	RoomTemp_204: FB_BACnetRM_AI := (Client:=Client,nObjectInstance:=52233);
	TempAdjust_204: FB_BACnetRM_AV := (Client:=Client,nObjectInstance:=52234);
	FilterSign_204: FB_BACnetRM_BI := (Client:=Client,nObjectInstance:=52235);
	FilterSignReset_204: FB_BACnetRM_BV := (Client:=Client,nObjectInstance:=52236);
	RemoteControlStart_204: FB_BACnetRM_BV := (Client:=Client,nObjectInstance:=52237);
	
	RemoteControlTempAdjust_204: FB_BACnetRM_BV := (Client:=Client,nObjectInstance:=52240);
	
	
	
	
	
	
	
	
	
	
	
	
	StartStopCommand_205: FB_BACnetRM_BO := (Client:=Client,nObjectInstance:=52481);
	StartStopStatus_205: FB_BACnetRM_BI := (Client:=Client,nObjectInstance:=52482);
	Alarm_205: FB_BACnetRM_BI := (Client:=Client,nObjectInstance:=52483);
	MalfunctionCode_205: FB_BACnetRM_MI := (Client:=Client,nObjectInstance:=52484);
	
	
	
	
	RoomTemp_205: FB_BACnetRM_AI := (Client:=Client,nObjectInstance:=52489);
	TempAdjust_205: FB_BACnetRM_AV := (Client:=Client,nObjectInstance:=52490);
	FilterSign_205: FB_BACnetRM_BI := (Client:=Client,nObjectInstance:=52491);
	FilterSignReset_205: FB_BACnetRM_BV := (Client:=Client,nObjectInstance:=52492);
	RemoteControlStart_205: FB_BACnetRM_BV := (Client:=Client,nObjectInstance:=52493);
	
	RemoteControlTempAdjust_205: FB_BACnetRM_BV := (Client:=Client,nObjectInstance:=52496);
	
	
	
	
	
	
	
	
	
	
	
	
	StartStopCommand_206: FB_BACnetRM_BO := (Client:=Client,nObjectInstance:=52737);
	StartStopStatus_206: FB_BACnetRM_BI := (Client:=Client,nObjectInstance:=52738);
	Alarm_206: FB_BACnetRM_BI := (Client:=Client,nObjectInstance:=52739);
	MalfunctionCode_206: FB_BACnetRM_MI := (Client:=Client,nObjectInstance:=52740);
	
	
	
	
	RoomTemp_206: FB_BACnetRM_AI := (Client:=Client,nObjectInstance:=52745);
	TempAdjust_206: FB_BACnetRM_AV := (Client:=Client,nObjectInstance:=52746);
	FilterSign_206: FB_BACnetRM_BI := (Client:=Client,nObjectInstance:=52747);
	FilterSignReset_206: FB_BACnetRM_BV := (Client:=Client,nObjectInstance:=52748);
	RemoteControlStart_206: FB_BACnetRM_BV := (Client:=Client,nObjectInstance:=52749);
	
	RemoteControlTempAdjust_206: FB_BACnetRM_BV := (Client:=Client,nObjectInstance:=52752);
	
	
	
	
	
	
	
	
	
	
	
	
	StartStopCommand_207: FB_BACnetRM_BO := (Client:=Client,nObjectInstance:=52993);
	StartStopStatus_207: FB_BACnetRM_BI := (Client:=Client,nObjectInstance:=52994);
	Alarm_207: FB_BACnetRM_BI := (Client:=Client,nObjectInstance:=52995);
	MalfunctionCode_207: FB_BACnetRM_MI := (Client:=Client,nObjectInstance:=52996);
	
	
	
	
	RoomTemp_207: FB_BACnetRM_AI := (Client:=Client,nObjectInstance:=53001);
	TempAdjust_207: FB_BACnetRM_AV := (Client:=Client,nObjectInstance:=53002);
	FilterSign_207: FB_BACnetRM_BI := (Client:=Client,nObjectInstance:=53003);
	FilterSignReset_207: FB_BACnetRM_BV := (Client:=Client,nObjectInstance:=53004);
	RemoteControlStart_207: FB_BACnetRM_BV := (Client:=Client,nObjectInstance:=53005);
	
	RemoteControlTempAdjust_207: FB_BACnetRM_BV := (Client:=Client,nObjectInstance:=53008);
	
	
	
	
	
	
	
	
	
	
	
	
	StartStopCommand_208: FB_BACnetRM_BO := (Client:=Client,nObjectInstance:=53249);
	StartStopStatus_208: FB_BACnetRM_BI := (Client:=Client,nObjectInstance:=53250);
	Alarm_208: FB_BACnetRM_BI := (Client:=Client,nObjectInstance:=53251);
	MalfunctionCode_208: FB_BACnetRM_MI := (Client:=Client,nObjectInstance:=53252);
	
	
	
	
	RoomTemp_208: FB_BACnetRM_AI := (Client:=Client,nObjectInstance:=53257);
	TempAdjust_208: FB_BACnetRM_AV := (Client:=Client,nObjectInstance:=53258);
	FilterSign_208: FB_BACnetRM_BI := (Client:=Client,nObjectInstance:=53259);
	FilterSignReset_208: FB_BACnetRM_BV := (Client:=Client,nObjectInstance:=53260);
	RemoteControlStart_208: FB_BACnetRM_BV := (Client:=Client,nObjectInstance:=53261);
	
	RemoteControlTempAdjust_208: FB_BACnetRM_BV := (Client:=Client,nObjectInstance:=53264);
	
	
	
	
	
	
	
	
	
	
	
	
	StartStopCommand_209: FB_BACnetRM_BO := (Client:=Client,nObjectInstance:=53505);
	StartStopStatus_209: FB_BACnetRM_BI := (Client:=Client,nObjectInstance:=53506);
	Alarm_209: FB_BACnetRM_BI := (Client:=Client,nObjectInstance:=53507);
	MalfunctionCode_209: FB_BACnetRM_MI := (Client:=Client,nObjectInstance:=53508);
	
	
	
	
	RoomTemp_209: FB_BACnetRM_AI := (Client:=Client,nObjectInstance:=53513);
	TempAdjust_209: FB_BACnetRM_AV := (Client:=Client,nObjectInstance:=53514);
	FilterSign_209: FB_BACnetRM_BI := (Client:=Client,nObjectInstance:=53515);
	FilterSignReset_209: FB_BACnetRM_BV := (Client:=Client,nObjectInstance:=53516);
	RemoteControlStart_209: FB_BACnetRM_BV := (Client:=Client,nObjectInstance:=53517);
	
	RemoteControlTempAdjust_209: FB_BACnetRM_BV := (Client:=Client,nObjectInstance:=53520);
	
	
	
	
	
	
	
	
	
	
	
	
	StartStopCommand_210: FB_BACnetRM_BO := (Client:=Client,nObjectInstance:=53761);
	StartStopStatus_210: FB_BACnetRM_BI := (Client:=Client,nObjectInstance:=53762);
	Alarm_210: FB_BACnetRM_BI := (Client:=Client,nObjectInstance:=53763);
	MalfunctionCode_210: FB_BACnetRM_MI := (Client:=Client,nObjectInstance:=53764);
	
	
	
	
	RoomTemp_210: FB_BACnetRM_AI := (Client:=Client,nObjectInstance:=53769);
	TempAdjust_210: FB_BACnetRM_AV := (Client:=Client,nObjectInstance:=53770);
	FilterSign_210: FB_BACnetRM_BI := (Client:=Client,nObjectInstance:=53771);
	FilterSignReset_210: FB_BACnetRM_BV := (Client:=Client,nObjectInstance:=53772);
	RemoteControlStart_210: FB_BACnetRM_BV := (Client:=Client,nObjectInstance:=53773);
	
	RemoteControlTempAdjust_210: FB_BACnetRM_BV := (Client:=Client,nObjectInstance:=53776);
	
	
	
	
	
	
	
	
	
	
	
	
	StartStopCommand_211: FB_BACnetRM_BO := (Client:=Client,nObjectInstance:=54017);
	StartStopStatus_211: FB_BACnetRM_BI := (Client:=Client,nObjectInstance:=54018);
	Alarm_211: FB_BACnetRM_BI := (Client:=Client,nObjectInstance:=54019);
	MalfunctionCode_211: FB_BACnetRM_MI := (Client:=Client,nObjectInstance:=54020);
	
	
	
	
	RoomTemp_211: FB_BACnetRM_AI := (Client:=Client,nObjectInstance:=54025);
	TempAdjust_211: FB_BACnetRM_AV := (Client:=Client,nObjectInstance:=54026);
	FilterSign_211: FB_BACnetRM_BI := (Client:=Client,nObjectInstance:=54027);
	FilterSignReset_211: FB_BACnetRM_BV := (Client:=Client,nObjectInstance:=54028);
	RemoteControlStart_211: FB_BACnetRM_BV := (Client:=Client,nObjectInstance:=54029);
	
	RemoteControlTempAdjust_211: FB_BACnetRM_BV := (Client:=Client,nObjectInstance:=54032);
	
	
	
	
	
	
	
	
	
	
	
	
	StartStopCommand_212: FB_BACnetRM_BO := (Client:=Client,nObjectInstance:=54273);
	StartStopStatus_212: FB_BACnetRM_BI := (Client:=Client,nObjectInstance:=54274);
	Alarm_212: FB_BACnetRM_BI := (Client:=Client,nObjectInstance:=54275);
	MalfunctionCode_212: FB_BACnetRM_MI := (Client:=Client,nObjectInstance:=54276);
	
	
	
	
	RoomTemp_212: FB_BACnetRM_AI := (Client:=Client,nObjectInstance:=54281);
	TempAdjust_212: FB_BACnetRM_AV := (Client:=Client,nObjectInstance:=54282);
	FilterSign_212: FB_BACnetRM_BI := (Client:=Client,nObjectInstance:=54283);
	FilterSignReset_212: FB_BACnetRM_BV := (Client:=Client,nObjectInstance:=54284);
	RemoteControlStart_212: FB_BACnetRM_BV := (Client:=Client,nObjectInstance:=54285);
	
	RemoteControlTempAdjust_212: FB_BACnetRM_BV := (Client:=Client,nObjectInstance:=54288);
	
	
	
	
	
	
	
	
	
	
	
	
	StartStopCommand_213: FB_BACnetRM_BO := (Client:=Client,nObjectInstance:=54529);
	StartStopStatus_213: FB_BACnetRM_BI := (Client:=Client,nObjectInstance:=54530);
	Alarm_213: FB_BACnetRM_BI := (Client:=Client,nObjectInstance:=54531);
	MalfunctionCode_213: FB_BACnetRM_MI := (Client:=Client,nObjectInstance:=54532);
	
	
	
	
	RoomTemp_213: FB_BACnetRM_AI := (Client:=Client,nObjectInstance:=54537);
	TempAdjust_213: FB_BACnetRM_AV := (Client:=Client,nObjectInstance:=54538);
	FilterSign_213: FB_BACnetRM_BI := (Client:=Client,nObjectInstance:=54539);
	FilterSignReset_213: FB_BACnetRM_BV := (Client:=Client,nObjectInstance:=54540);
	RemoteControlStart_213: FB_BACnetRM_BV := (Client:=Client,nObjectInstance:=54541);
	
	RemoteControlTempAdjust_213: FB_BACnetRM_BV := (Client:=Client,nObjectInstance:=54544);
	
	
	
	
	
	
	
	
	
	
	
	
	StartStopCommand_214: FB_BACnetRM_BO := (Client:=Client,nObjectInstance:=54785);
	StartStopStatus_214: FB_BACnetRM_BI := (Client:=Client,nObjectInstance:=54786);
	Alarm_214: FB_BACnetRM_BI := (Client:=Client,nObjectInstance:=54787);
	MalfunctionCode_214: FB_BACnetRM_MI := (Client:=Client,nObjectInstance:=54788);
	
	
	
	
	RoomTemp_214: FB_BACnetRM_AI := (Client:=Client,nObjectInstance:=54793);
	TempAdjust_214: FB_BACnetRM_AV := (Client:=Client,nObjectInstance:=54794);
	FilterSign_214: FB_BACnetRM_BI := (Client:=Client,nObjectInstance:=54795);
	FilterSignReset_214: FB_BACnetRM_BV := (Client:=Client,nObjectInstance:=54796);
	RemoteControlStart_214: FB_BACnetRM_BV := (Client:=Client,nObjectInstance:=54797);
	
	RemoteControlTempAdjust_214: FB_BACnetRM_BV := (Client:=Client,nObjectInstance:=54800);
	
	
	
	
	
	
	
	
	
	
	
	
	StartStopCommand_215: FB_BACnetRM_BO := (Client:=Client,nObjectInstance:=55041);
	StartStopStatus_215: FB_BACnetRM_BI := (Client:=Client,nObjectInstance:=55042);
	Alarm_215: FB_BACnetRM_BI := (Client:=Client,nObjectInstance:=55043);
	MalfunctionCode_215: FB_BACnetRM_MI := (Client:=Client,nObjectInstance:=55044);
	
	
	
	
	RoomTemp_215: FB_BACnetRM_AI := (Client:=Client,nObjectInstance:=55049);
	TempAdjust_215: FB_BACnetRM_AV := (Client:=Client,nObjectInstance:=55050);
	FilterSign_215: FB_BACnetRM_BI := (Client:=Client,nObjectInstance:=55051);
	FilterSignReset_215: FB_BACnetRM_BV := (Client:=Client,nObjectInstance:=55052);
	RemoteControlStart_215: FB_BACnetRM_BV := (Client:=Client,nObjectInstance:=55053);
	
	RemoteControlTempAdjust_215: FB_BACnetRM_BV := (Client:=Client,nObjectInstance:=55056);
	
	
	
	
	
	
	
	
	
	
	
	
	StartStopCommand_216: FB_BACnetRM_BO := (Client:=Client,nObjectInstance:=55297);
	StartStopStatus_216: FB_BACnetRM_BI := (Client:=Client,nObjectInstance:=55298);
	Alarm_216: FB_BACnetRM_BI := (Client:=Client,nObjectInstance:=55299);
	MalfunctionCode_216: FB_BACnetRM_MI := (Client:=Client,nObjectInstance:=55300);
	
	
	
	
	RoomTemp_216: FB_BACnetRM_AI := (Client:=Client,nObjectInstance:=55305);
	TempAdjust_216: FB_BACnetRM_AV := (Client:=Client,nObjectInstance:=55306);
	FilterSign_216: FB_BACnetRM_BI := (Client:=Client,nObjectInstance:=55307);
	FilterSignReset_216: FB_BACnetRM_BV := (Client:=Client,nObjectInstance:=55308);
	RemoteControlStart_216: FB_BACnetRM_BV := (Client:=Client,nObjectInstance:=55309);
	
	RemoteControlTempAdjust_216: FB_BACnetRM_BV := (Client:=Client,nObjectInstance:=55312);
	
	
	
	
	
	
	
	
	
	
	
	
	StartStopCommand_217: FB_BACnetRM_BO := (Client:=Client,nObjectInstance:=55553);
	StartStopStatus_217: FB_BACnetRM_BI := (Client:=Client,nObjectInstance:=55554);
	Alarm_217: FB_BACnetRM_BI := (Client:=Client,nObjectInstance:=55555);
	MalfunctionCode_217: FB_BACnetRM_MI := (Client:=Client,nObjectInstance:=55556);
	
	
	
	
	RoomTemp_217: FB_BACnetRM_AI := (Client:=Client,nObjectInstance:=55561);
	TempAdjust_217: FB_BACnetRM_AV := (Client:=Client,nObjectInstance:=55562);
	FilterSign_217: FB_BACnetRM_BI := (Client:=Client,nObjectInstance:=55563);
	FilterSignReset_217: FB_BACnetRM_BV := (Client:=Client,nObjectInstance:=55564);
	RemoteControlStart_217: FB_BACnetRM_BV := (Client:=Client,nObjectInstance:=55565);
	
	RemoteControlTempAdjust_217: FB_BACnetRM_BV := (Client:=Client,nObjectInstance:=55568);
	
	
	
	
	
	
	
	
	
	
	
	
	StartStopCommand_224: FB_BACnetRM_BO := (Client:=Client,nObjectInstance:=57345);
	StartStopStatus_224: FB_BACnetRM_BI := (Client:=Client,nObjectInstance:=57346);
	Alarm_224: FB_BACnetRM_BI := (Client:=Client,nObjectInstance:=57347);
	MalfunctionCode_224: FB_BACnetRM_MI := (Client:=Client,nObjectInstance:=57348);
	
	
	
	
	RoomTemp_224: FB_BACnetRM_AI := (Client:=Client,nObjectInstance:=57353);
	TempAdjust_224: FB_BACnetRM_AV := (Client:=Client,nObjectInstance:=57354);
	FilterSign_224: FB_BACnetRM_BI := (Client:=Client,nObjectInstance:=57355);
	FilterSignReset_224: FB_BACnetRM_BV := (Client:=Client,nObjectInstance:=57356);
	RemoteControlStart_224: FB_BACnetRM_BV := (Client:=Client,nObjectInstance:=57357);
	
	RemoteControlTempAdjust_224: FB_BACnetRM_BV := (Client:=Client,nObjectInstance:=57360);
	
	
	
	
	
	
	
	
	
	
	
	
	StartStopCommand_225: FB_BACnetRM_BO := (Client:=Client,nObjectInstance:=57601);
	StartStopStatus_225: FB_BACnetRM_BI := (Client:=Client,nObjectInstance:=57602);
	Alarm_225: FB_BACnetRM_BI := (Client:=Client,nObjectInstance:=57603);
	MalfunctionCode_225: FB_BACnetRM_MI := (Client:=Client,nObjectInstance:=57604);
	
	
	
	
	RoomTemp_225: FB_BACnetRM_AI := (Client:=Client,nObjectInstance:=57609);
	TempAdjust_225: FB_BACnetRM_AV := (Client:=Client,nObjectInstance:=57610);
	FilterSign_225: FB_BACnetRM_BI := (Client:=Client,nObjectInstance:=57611);
	FilterSignReset_225: FB_BACnetRM_BV := (Client:=Client,nObjectInstance:=57612);
	RemoteControlStart_225: FB_BACnetRM_BV := (Client:=Client,nObjectInstance:=57613);
	
	RemoteControlTempAdjust_225: FB_BACnetRM_BV := (Client:=Client,nObjectInstance:=57616);
	
	
	
	
	
	
	
	
	
	
	
	
	StartStopCommand_226: FB_BACnetRM_BO := (Client:=Client,nObjectInstance:=57857);
	StartStopStatus_226: FB_BACnetRM_BI := (Client:=Client,nObjectInstance:=57858);
	Alarm_226: FB_BACnetRM_BI := (Client:=Client,nObjectInstance:=57859);
	MalfunctionCode_226: FB_BACnetRM_MI := (Client:=Client,nObjectInstance:=57860);
	
	
	
	
	RoomTemp_226: FB_BACnetRM_AI := (Client:=Client,nObjectInstance:=57865);
	TempAdjust_226: FB_BACnetRM_AV := (Client:=Client,nObjectInstance:=57866);
	FilterSign_226: FB_BACnetRM_BI := (Client:=Client,nObjectInstance:=57867);
	FilterSignReset_226: FB_BACnetRM_BV := (Client:=Client,nObjectInstance:=57868);
	RemoteControlStart_226: FB_BACnetRM_BV := (Client:=Client,nObjectInstance:=57869);
	
	RemoteControlTempAdjust_226: FB_BACnetRM_BV := (Client:=Client,nObjectInstance:=57872);
	
	
	
	
	
	
	
	
	
	
	
	
	StartStopCommand_227: FB_BACnetRM_BO := (Client:=Client,nObjectInstance:=58113);
	StartStopStatus_227: FB_BACnetRM_BI := (Client:=Client,nObjectInstance:=58114);
	Alarm_227: FB_BACnetRM_BI := (Client:=Client,nObjectInstance:=58115);
	MalfunctionCode_227: FB_BACnetRM_MI := (Client:=Client,nObjectInstance:=58116);
	
	
	
	
	RoomTemp_227: FB_BACnetRM_AI := (Client:=Client,nObjectInstance:=58121);
	TempAdjust_227: FB_BACnetRM_AV := (Client:=Client,nObjectInstance:=58122);
	FilterSign_227: FB_BACnetRM_BI := (Client:=Client,nObjectInstance:=58123);
	FilterSignReset_227: FB_BACnetRM_BV := (Client:=Client,nObjectInstance:=58124);
	RemoteControlStart_227: FB_BACnetRM_BV := (Client:=Client,nObjectInstance:=58125);
	
	RemoteControlTempAdjust_227: FB_BACnetRM_BV := (Client:=Client,nObjectInstance:=58128);
	
	
	
	
	
	
	
	
	
	
	
	
	StartStopCommand_240: FB_BACnetRM_BO := (Client:=Client,nObjectInstance:=61441);
	StartStopStatus_240: FB_BACnetRM_BI := (Client:=Client,nObjectInstance:=61442);
	Alarm_240: FB_BACnetRM_BI := (Client:=Client,nObjectInstance:=61443);
	MalfunctionCode_240: FB_BACnetRM_MI := (Client:=Client,nObjectInstance:=61444);
	
	
	
	
	RoomTemp_240: FB_BACnetRM_AI := (Client:=Client,nObjectInstance:=61449);
	TempAdjust_240: FB_BACnetRM_AV := (Client:=Client,nObjectInstance:=61450);
	FilterSign_240: FB_BACnetRM_BI := (Client:=Client,nObjectInstance:=61451);
	FilterSignReset_240: FB_BACnetRM_BV := (Client:=Client,nObjectInstance:=61452);
	RemoteControlStart_240: FB_BACnetRM_BV := (Client:=Client,nObjectInstance:=61453);
	
	RemoteControlTempAdjust_240: FB_BACnetRM_BV := (Client:=Client,nObjectInstance:=61456);
	
	
	
	
	
	
	
	
	
	
	
	
	StartStopCommand_241: FB_BACnetRM_BO := (Client:=Client,nObjectInstance:=61697);
	StartStopStatus_241: FB_BACnetRM_BI := (Client:=Client,nObjectInstance:=61698);
	Alarm_241: FB_BACnetRM_BI := (Client:=Client,nObjectInstance:=61699);
	MalfunctionCode_241: FB_BACnetRM_MI := (Client:=Client,nObjectInstance:=61700);
	
	
	
	
	RoomTemp_241: FB_BACnetRM_AI := (Client:=Client,nObjectInstance:=61705);
	TempAdjust_241: FB_BACnetRM_AV := (Client:=Client,nObjectInstance:=61706);
	FilterSign_241: FB_BACnetRM_BI := (Client:=Client,nObjectInstance:=61707);
	FilterSignReset_241: FB_BACnetRM_BV := (Client:=Client,nObjectInstance:=61708);
	RemoteControlStart_241: FB_BACnetRM_BV := (Client:=Client,nObjectInstance:=61709);
	
	RemoteControlTempAdjust_241: FB_BACnetRM_BV := (Client:=Client,nObjectInstance:=61712);
	
	
	
	
	
	
	
	
	
	
	
	
	CL_Rejection_000: FB_BACnetRM_BV := (Client:=Client,nObjectInstance:=17);
	SystemForcedOff_000: FB_BACnetRM_BV := (Client:=Client,nObjectInstance:=21);
	CL_Rejection_064: FB_BACnetRM_BV := (Client:=Client,nObjectInstance:=16401);
	SystemForcedOff_064: FB_BACnetRM_BV := (Client:=Client,nObjectInstance:=16405);
	CL_Rejection_128: FB_BACnetRM_BV := (Client:=Client,nObjectInstance:=32785);
	SystemForcedOff_128: FB_BACnetRM_BV := (Client:=Client,nObjectInstance:=32789);
	CL_Rejection_192: FB_BACnetRM_BV := (Client:=Client,nObjectInstance:=49169);
	SystemForcedOff_192: FB_BACnetRM_BV := (Client:=Client,nObjectInstance:=49173);
END_VAR

Client();
DAIKIN_MasterStation_III_No_1();
StartStopCommand_000();
StartStopStatus_000();
Alarm_000();
MalfunctionCode_000();




RoomTemp_000();
TempAdjust_000();
FilterSign_000();
FilterSignReset_000();
RemoteControlStart_000();

RemoteControlTempAdjust_000();












StartStopCommand_001();
StartStopStatus_001();
Alarm_001();
MalfunctionCode_001();




RoomTemp_001();
TempAdjust_001();
FilterSign_001();
FilterSignReset_001();
RemoteControlStart_001();

RemoteControlTempAdjust_001();












StartStopCommand_002();
StartStopStatus_002();
Alarm_002();
MalfunctionCode_002();




RoomTemp_002();
TempAdjust_002();
FilterSign_002();
FilterSignReset_002();
RemoteControlStart_002();

RemoteControlTempAdjust_002();












StartStopCommand_003();
StartStopStatus_003();
Alarm_003();
MalfunctionCode_003();




RoomTemp_003();
TempAdjust_003();
FilterSign_003();
FilterSignReset_003();
RemoteControlStart_003();

RemoteControlTempAdjust_003();












StartStopCommand_004();
StartStopStatus_004();
Alarm_004();
MalfunctionCode_004();




RoomTemp_004();
TempAdjust_004();
FilterSign_004();
FilterSignReset_004();
RemoteControlStart_004();

RemoteControlTempAdjust_004();












StartStopCommand_005();
StartStopStatus_005();
Alarm_005();
MalfunctionCode_005();




RoomTemp_005();
TempAdjust_005();
FilterSign_005();
FilterSignReset_005();
RemoteControlStart_005();

RemoteControlTempAdjust_005();












StartStopCommand_006();
StartStopStatus_006();
Alarm_006();
MalfunctionCode_006();




RoomTemp_006();
TempAdjust_006();
FilterSign_006();
FilterSignReset_006();
RemoteControlStart_006();

RemoteControlTempAdjust_006();












StartStopCommand_007();
StartStopStatus_007();
Alarm_007();
MalfunctionCode_007();




RoomTemp_007();
TempAdjust_007();
FilterSign_007();
FilterSignReset_007();
RemoteControlStart_007();

RemoteControlTempAdjust_007();












StartStopCommand_008();
StartStopStatus_008();
Alarm_008();
MalfunctionCode_008();




RoomTemp_008();
TempAdjust_008();
FilterSign_008();
FilterSignReset_008();
RemoteControlStart_008();

RemoteControlTempAdjust_008();












StartStopCommand_009();
StartStopStatus_009();
Alarm_009();
MalfunctionCode_009();




RoomTemp_009();
TempAdjust_009();
FilterSign_009();
FilterSignReset_009();
RemoteControlStart_009();

RemoteControlTempAdjust_009();












StartStopCommand_010();
StartStopStatus_010();
Alarm_010();
MalfunctionCode_010();




RoomTemp_010();
TempAdjust_010();
FilterSign_010();
FilterSignReset_010();
RemoteControlStart_010();

RemoteControlTempAdjust_010();












StartStopCommand_011();
StartStopStatus_011();
Alarm_011();
MalfunctionCode_011();




RoomTemp_011();
TempAdjust_011();
FilterSign_011();
FilterSignReset_011();
RemoteControlStart_011();

RemoteControlTempAdjust_011();












StartStopCommand_012();
StartStopStatus_012();
Alarm_012();
MalfunctionCode_012();




RoomTemp_012();
TempAdjust_012();
FilterSign_012();
FilterSignReset_012();
RemoteControlStart_012();

RemoteControlTempAdjust_012();












StartStopCommand_013();
StartStopStatus_013();
Alarm_013();
MalfunctionCode_013();




RoomTemp_013();
TempAdjust_013();
FilterSign_013();
FilterSignReset_013();
RemoteControlStart_013();

RemoteControlTempAdjust_013();












StartStopCommand_014();
StartStopStatus_014();
Alarm_014();
MalfunctionCode_014();




RoomTemp_014();
TempAdjust_014();
FilterSign_014();
FilterSignReset_014();
RemoteControlStart_014();

RemoteControlTempAdjust_014();












StartStopCommand_015();
StartStopStatus_015();
Alarm_015();
MalfunctionCode_015();




RoomTemp_015();
TempAdjust_015();
FilterSign_015();
FilterSignReset_015();
RemoteControlStart_015();

RemoteControlTempAdjust_015();












StartStopCommand_016();
StartStopStatus_016();
Alarm_016();
MalfunctionCode_016();




RoomTemp_016();
TempAdjust_016();
FilterSign_016();
FilterSignReset_016();
RemoteControlStart_016();

RemoteControlTempAdjust_016();












StartStopCommand_017();
StartStopStatus_017();
Alarm_017();
MalfunctionCode_017();




RoomTemp_017();
TempAdjust_017();
FilterSign_017();
FilterSignReset_017();
RemoteControlStart_017();

RemoteControlTempAdjust_017();












StartStopCommand_018();
StartStopStatus_018();
Alarm_018();
MalfunctionCode_018();




RoomTemp_018();
TempAdjust_018();
FilterSign_018();
FilterSignReset_018();
RemoteControlStart_018();

RemoteControlTempAdjust_018();












StartStopCommand_019();
StartStopStatus_019();
Alarm_019();
MalfunctionCode_019();




RoomTemp_019();
TempAdjust_019();
FilterSign_019();
FilterSignReset_019();
RemoteControlStart_019();

RemoteControlTempAdjust_019();












StartStopCommand_020();
StartStopStatus_020();
Alarm_020();
MalfunctionCode_020();




RoomTemp_020();
TempAdjust_020();
FilterSign_020();
FilterSignReset_020();
RemoteControlStart_020();

RemoteControlTempAdjust_020();












StartStopCommand_021();
StartStopStatus_021();
Alarm_021();
MalfunctionCode_021();




RoomTemp_021();
TempAdjust_021();
FilterSign_021();
FilterSignReset_021();
RemoteControlStart_021();

RemoteControlTempAdjust_021();












StartStopCommand_022();
StartStopStatus_022();
Alarm_022();
MalfunctionCode_022();




RoomTemp_022();
TempAdjust_022();
FilterSign_022();
FilterSignReset_022();
RemoteControlStart_022();

RemoteControlTempAdjust_022();












StartStopCommand_023();
StartStopStatus_023();
Alarm_023();
MalfunctionCode_023();




RoomTemp_023();
TempAdjust_023();
FilterSign_023();
FilterSignReset_023();
RemoteControlStart_023();

RemoteControlTempAdjust_023();












StartStopCommand_024();
StartStopStatus_024();
Alarm_024();
MalfunctionCode_024();




RoomTemp_024();
TempAdjust_024();
FilterSign_024();
FilterSignReset_024();
RemoteControlStart_024();

RemoteControlTempAdjust_024();












StartStopCommand_025();
StartStopStatus_025();
Alarm_025();
MalfunctionCode_025();




RoomTemp_025();
TempAdjust_025();
FilterSign_025();
FilterSignReset_025();
RemoteControlStart_025();

RemoteControlTempAdjust_025();












StartStopCommand_026();
StartStopStatus_026();
Alarm_026();
MalfunctionCode_026();




RoomTemp_026();
TempAdjust_026();
FilterSign_026();
FilterSignReset_026();
RemoteControlStart_026();

RemoteControlTempAdjust_026();












StartStopCommand_027();
StartStopStatus_027();
Alarm_027();
MalfunctionCode_027();




RoomTemp_027();
TempAdjust_027();
FilterSign_027();
FilterSignReset_027();
RemoteControlStart_027();

RemoteControlTempAdjust_027();












StartStopCommand_028();
StartStopStatus_028();
Alarm_028();
MalfunctionCode_028();




RoomTemp_028();
TempAdjust_028();
FilterSign_028();
FilterSignReset_028();
RemoteControlStart_028();

RemoteControlTempAdjust_028();












StartStopCommand_029();
StartStopStatus_029();
Alarm_029();
MalfunctionCode_029();




RoomTemp_029();
TempAdjust_029();
FilterSign_029();
FilterSignReset_029();
RemoteControlStart_029();

RemoteControlTempAdjust_029();












StartStopCommand_030();
StartStopStatus_030();
Alarm_030();
MalfunctionCode_030();




RoomTemp_030();
TempAdjust_030();
FilterSign_030();
FilterSignReset_030();
RemoteControlStart_030();

RemoteControlTempAdjust_030();












StartStopCommand_031();
StartStopStatus_031();
Alarm_031();
MalfunctionCode_031();




RoomTemp_031();
TempAdjust_031();
FilterSign_031();
FilterSignReset_031();
RemoteControlStart_031();

RemoteControlTempAdjust_031();












StartStopCommand_032();
StartStopStatus_032();
Alarm_032();
MalfunctionCode_032();




RoomTemp_032();
TempAdjust_032();
FilterSign_032();
FilterSignReset_032();
RemoteControlStart_032();

RemoteControlTempAdjust_032();












StartStopCommand_033();
StartStopStatus_033();
Alarm_033();
MalfunctionCode_033();




RoomTemp_033();
TempAdjust_033();
FilterSign_033();
FilterSignReset_033();
RemoteControlStart_033();

RemoteControlTempAdjust_033();












StartStopCommand_034();
StartStopStatus_034();
Alarm_034();
MalfunctionCode_034();




RoomTemp_034();
TempAdjust_034();
FilterSign_034();
FilterSignReset_034();
RemoteControlStart_034();

RemoteControlTempAdjust_034();












StartStopCommand_035();
StartStopStatus_035();
Alarm_035();
MalfunctionCode_035();




RoomTemp_035();
TempAdjust_035();
FilterSign_035();
FilterSignReset_035();
RemoteControlStart_035();

RemoteControlTempAdjust_035();












StartStopCommand_036();
StartStopStatus_036();
Alarm_036();
MalfunctionCode_036();




RoomTemp_036();
TempAdjust_036();
FilterSign_036();
FilterSignReset_036();
RemoteControlStart_036();

RemoteControlTempAdjust_036();












StartStopCommand_037();
StartStopStatus_037();
Alarm_037();
MalfunctionCode_037();




RoomTemp_037();
TempAdjust_037();
FilterSign_037();
FilterSignReset_037();
RemoteControlStart_037();

RemoteControlTempAdjust_037();












StartStopCommand_038();
StartStopStatus_038();
Alarm_038();
MalfunctionCode_038();




RoomTemp_038();
TempAdjust_038();
FilterSign_038();
FilterSignReset_038();
RemoteControlStart_038();

RemoteControlTempAdjust_038();












StartStopCommand_039();
StartStopStatus_039();
Alarm_039();
MalfunctionCode_039();




RoomTemp_039();
TempAdjust_039();
FilterSign_039();
FilterSignReset_039();
RemoteControlStart_039();

RemoteControlTempAdjust_039();












StartStopCommand_041();
StartStopStatus_041();
Alarm_041();
MalfunctionCode_041();




RoomTemp_041();
TempAdjust_041();
FilterSign_041();
FilterSignReset_041();
RemoteControlStart_041();

RemoteControlTempAdjust_041();












StartStopCommand_042();
StartStopStatus_042();
Alarm_042();
MalfunctionCode_042();




RoomTemp_042();
TempAdjust_042();
FilterSign_042();
FilterSignReset_042();
RemoteControlStart_042();

RemoteControlTempAdjust_042();












StartStopCommand_043();
StartStopStatus_043();
Alarm_043();
MalfunctionCode_043();




RoomTemp_043();
TempAdjust_043();
FilterSign_043();
FilterSignReset_043();
RemoteControlStart_043();

RemoteControlTempAdjust_043();












//StartStopCommand_044();
//StartStopStatus_044();
//Alarm_044();
//MalfunctionCode_044();




//RoomTemp_044();
//TempAdjust_044();
//FilterSign_044();
//FilterSignReset_044();
//RemoteControlStart_044();
//
//RemoteControlTempAdjust_044();

//










StartStopCommand_045();
StartStopStatus_045();
Alarm_045();
MalfunctionCode_045();




RoomTemp_045();
TempAdjust_045();
FilterSign_045();
FilterSignReset_045();
RemoteControlStart_045();

RemoteControlTempAdjust_045();












StartStopCommand_046();
StartStopStatus_046();
Alarm_046();
MalfunctionCode_046();




RoomTemp_046();
TempAdjust_046();
FilterSign_046();
FilterSignReset_046();
RemoteControlStart_046();

RemoteControlTempAdjust_046();












//StartStopCommand_048();
//StartStopStatus_048();
//Alarm_048();
//MalfunctionCode_048();




//RoomTemp_048();
//TempAdjust_048();
//FilterSign_048();
//FilterSignReset_048();
//RemoteControlStart_048();
//
//RemoteControlTempAdjust_048();

//










StartStopCommand_049();
StartStopStatus_049();
Alarm_049();
MalfunctionCode_049();




RoomTemp_049();
TempAdjust_049();
FilterSign_049();
FilterSignReset_049();
RemoteControlStart_049();

RemoteControlTempAdjust_049();












StartStopCommand_064();
StartStopStatus_064();
Alarm_064();
MalfunctionCode_064();




RoomTemp_064();
TempAdjust_064();
FilterSign_064();
FilterSignReset_064();
RemoteControlStart_064();

RemoteControlTempAdjust_064();












StartStopCommand_065();
StartStopStatus_065();
Alarm_065();
MalfunctionCode_065();




RoomTemp_065();
TempAdjust_065();
FilterSign_065();
FilterSignReset_065();
RemoteControlStart_065();

RemoteControlTempAdjust_065();












StartStopCommand_066();
StartStopStatus_066();
Alarm_066();
MalfunctionCode_066();




RoomTemp_066();
TempAdjust_066();
FilterSign_066();
FilterSignReset_066();
RemoteControlStart_066();

RemoteControlTempAdjust_066();












StartStopCommand_067();
StartStopStatus_067();
Alarm_067();
MalfunctionCode_067();




RoomTemp_067();
TempAdjust_067();
FilterSign_067();
FilterSignReset_067();
RemoteControlStart_067();

RemoteControlTempAdjust_067();












StartStopCommand_068();
StartStopStatus_068();
Alarm_068();
MalfunctionCode_068();




RoomTemp_068();
TempAdjust_068();
FilterSign_068();
FilterSignReset_068();
RemoteControlStart_068();

RemoteControlTempAdjust_068();












StartStopCommand_069();
StartStopStatus_069();
Alarm_069();
MalfunctionCode_069();




RoomTemp_069();
TempAdjust_069();
FilterSign_069();
FilterSignReset_069();
RemoteControlStart_069();

RemoteControlTempAdjust_069();












StartStopCommand_070();
StartStopStatus_070();
Alarm_070();
MalfunctionCode_070();




RoomTemp_070();
TempAdjust_070();
FilterSign_070();
FilterSignReset_070();
RemoteControlStart_070();

RemoteControlTempAdjust_070();












StartStopCommand_071();
StartStopStatus_071();
Alarm_071();
MalfunctionCode_071();




RoomTemp_071();
TempAdjust_071();
FilterSign_071();
FilterSignReset_071();
RemoteControlStart_071();

RemoteControlTempAdjust_071();












StartStopCommand_072();
StartStopStatus_072();
Alarm_072();
MalfunctionCode_072();




RoomTemp_072();
TempAdjust_072();
FilterSign_072();
FilterSignReset_072();
RemoteControlStart_072();

RemoteControlTempAdjust_072();












StartStopCommand_073();
StartStopStatus_073();
Alarm_073();
MalfunctionCode_073();




RoomTemp_073();
TempAdjust_073();
FilterSign_073();
FilterSignReset_073();
RemoteControlStart_073();

RemoteControlTempAdjust_073();












StartStopCommand_074();
StartStopStatus_074();
Alarm_074();
MalfunctionCode_074();




RoomTemp_074();
TempAdjust_074();
FilterSign_074();
FilterSignReset_074();
RemoteControlStart_074();

RemoteControlTempAdjust_074();












StartStopCommand_075();
StartStopStatus_075();
Alarm_075();
MalfunctionCode_075();




RoomTemp_075();
TempAdjust_075();
FilterSign_075();
FilterSignReset_075();
RemoteControlStart_075();

RemoteControlTempAdjust_075();












StartStopCommand_076();
StartStopStatus_076();
Alarm_076();
MalfunctionCode_076();




RoomTemp_076();
TempAdjust_076();
FilterSign_076();
FilterSignReset_076();
RemoteControlStart_076();

RemoteControlTempAdjust_076();












StartStopCommand_077();
StartStopStatus_077();
Alarm_077();
MalfunctionCode_077();




RoomTemp_077();
TempAdjust_077();
FilterSign_077();
FilterSignReset_077();
RemoteControlStart_077();

RemoteControlTempAdjust_077();












StartStopCommand_078();
StartStopStatus_078();
Alarm_078();
MalfunctionCode_078();




RoomTemp_078();
TempAdjust_078();
FilterSign_078();
FilterSignReset_078();
RemoteControlStart_078();

RemoteControlTempAdjust_078();












StartStopCommand_079();
StartStopStatus_079();
Alarm_079();
MalfunctionCode_079();




RoomTemp_079();
TempAdjust_079();
FilterSign_079();
FilterSignReset_079();
RemoteControlStart_079();

RemoteControlTempAdjust_079();












StartStopCommand_080();
StartStopStatus_080();
Alarm_080();
MalfunctionCode_080();




RoomTemp_080();
TempAdjust_080();
FilterSign_080();
FilterSignReset_080();
RemoteControlStart_080();

RemoteControlTempAdjust_080();












StartStopCommand_081();
StartStopStatus_081();
Alarm_081();
MalfunctionCode_081();




RoomTemp_081();
TempAdjust_081();
FilterSign_081();
FilterSignReset_081();
RemoteControlStart_081();

RemoteControlTempAdjust_081();












StartStopCommand_082();
StartStopStatus_082();
Alarm_082();
MalfunctionCode_082();




RoomTemp_082();
TempAdjust_082();
FilterSign_082();
FilterSignReset_082();
RemoteControlStart_082();

RemoteControlTempAdjust_082();












StartStopCommand_083();
StartStopStatus_083();
Alarm_083();
MalfunctionCode_083();




RoomTemp_083();
TempAdjust_083();
FilterSign_083();
FilterSignReset_083();
RemoteControlStart_083();

RemoteControlTempAdjust_083();












StartStopCommand_084();
StartStopStatus_084();
Alarm_084();
MalfunctionCode_084();




RoomTemp_084();
TempAdjust_084();
FilterSign_084();
FilterSignReset_084();
RemoteControlStart_084();

RemoteControlTempAdjust_084();












StartStopCommand_085();
StartStopStatus_085();
Alarm_085();
MalfunctionCode_085();




RoomTemp_085();
TempAdjust_085();
FilterSign_085();
FilterSignReset_085();
RemoteControlStart_085();

RemoteControlTempAdjust_085();












StartStopCommand_096();
StartStopStatus_096();
Alarm_096();
MalfunctionCode_096();




RoomTemp_096();
TempAdjust_096();
FilterSign_096();
FilterSignReset_096();
RemoteControlStart_096();

RemoteControlTempAdjust_096();












StartStopCommand_097();
StartStopStatus_097();
Alarm_097();
MalfunctionCode_097();




RoomTemp_097();
TempAdjust_097();
FilterSign_097();
FilterSignReset_097();
RemoteControlStart_097();

RemoteControlTempAdjust_097();












StartStopCommand_098();
StartStopStatus_098();
Alarm_098();
MalfunctionCode_098();




RoomTemp_098();
TempAdjust_098();
FilterSign_098();
FilterSignReset_098();
RemoteControlStart_098();

RemoteControlTempAdjust_098();












StartStopCommand_099();
StartStopStatus_099();
Alarm_099();
MalfunctionCode_099();




RoomTemp_099();
TempAdjust_099();
FilterSign_099();
FilterSignReset_099();
RemoteControlStart_099();

RemoteControlTempAdjust_099();












StartStopCommand_100();
StartStopStatus_100();
Alarm_100();
MalfunctionCode_100();




RoomTemp_100();
TempAdjust_100();
FilterSign_100();
FilterSignReset_100();
RemoteControlStart_100();

RemoteControlTempAdjust_100();












StartStopCommand_101();
StartStopStatus_101();
Alarm_101();
MalfunctionCode_101();




RoomTemp_101();
TempAdjust_101();
FilterSign_101();
FilterSignReset_101();
RemoteControlStart_101();

RemoteControlTempAdjust_101();












StartStopCommand_102();
StartStopStatus_102();
Alarm_102();
MalfunctionCode_102();




RoomTemp_102();
TempAdjust_102();
FilterSign_102();
FilterSignReset_102();
RemoteControlStart_102();

RemoteControlTempAdjust_102();












StartStopCommand_103();
StartStopStatus_103();
Alarm_103();
MalfunctionCode_103();




RoomTemp_103();
TempAdjust_103();
FilterSign_103();
FilterSignReset_103();
RemoteControlStart_103();

RemoteControlTempAdjust_103();












StartStopCommand_104();
StartStopStatus_104();
Alarm_104();
MalfunctionCode_104();




RoomTemp_104();
TempAdjust_104();
FilterSign_104();
FilterSignReset_104();
RemoteControlStart_104();

RemoteControlTempAdjust_104();












StartStopCommand_105();
StartStopStatus_105();
Alarm_105();
MalfunctionCode_105();




RoomTemp_105();
TempAdjust_105();
FilterSign_105();
FilterSignReset_105();
RemoteControlStart_105();

RemoteControlTempAdjust_105();












StartStopCommand_128();
StartStopStatus_128();
Alarm_128();
MalfunctionCode_128();




RoomTemp_128();
TempAdjust_128();
FilterSign_128();
FilterSignReset_128();
RemoteControlStart_128();

RemoteControlTempAdjust_128();












StartStopCommand_129();
StartStopStatus_129();
Alarm_129();
MalfunctionCode_129();




RoomTemp_129();
TempAdjust_129();
FilterSign_129();
FilterSignReset_129();
RemoteControlStart_129();

RemoteControlTempAdjust_129();












StartStopCommand_130();
StartStopStatus_130();
Alarm_130();
MalfunctionCode_130();




RoomTemp_130();
TempAdjust_130();
FilterSign_130();
FilterSignReset_130();
RemoteControlStart_130();

RemoteControlTempAdjust_130();












StartStopCommand_131();
StartStopStatus_131();
Alarm_131();
MalfunctionCode_131();




RoomTemp_131();
TempAdjust_131();
FilterSign_131();
FilterSignReset_131();
RemoteControlStart_131();

RemoteControlTempAdjust_131();












StartStopCommand_132();
StartStopStatus_132();
Alarm_132();
MalfunctionCode_132();




RoomTemp_132();
TempAdjust_132();
FilterSign_132();
FilterSignReset_132();
RemoteControlStart_132();

RemoteControlTempAdjust_132();












StartStopCommand_133();
StartStopStatus_133();
Alarm_133();
MalfunctionCode_133();




RoomTemp_133();
TempAdjust_133();
FilterSign_133();
FilterSignReset_133();
RemoteControlStart_133();

RemoteControlTempAdjust_133();












StartStopCommand_134();
StartStopStatus_134();
Alarm_134();
MalfunctionCode_134();




RoomTemp_134();
TempAdjust_134();
FilterSign_134();
FilterSignReset_134();
RemoteControlStart_134();

RemoteControlTempAdjust_134();












StartStopCommand_135();
StartStopStatus_135();
Alarm_135();
MalfunctionCode_135();




RoomTemp_135();
TempAdjust_135();
FilterSign_135();
FilterSignReset_135();
RemoteControlStart_135();

RemoteControlTempAdjust_135();












StartStopCommand_136();
StartStopStatus_136();
Alarm_136();
MalfunctionCode_136();




RoomTemp_136();
TempAdjust_136();
FilterSign_136();
FilterSignReset_136();
RemoteControlStart_136();

RemoteControlTempAdjust_136();












StartStopCommand_137();
StartStopStatus_137();
Alarm_137();
MalfunctionCode_137();




RoomTemp_137();
TempAdjust_137();
FilterSign_137();
FilterSignReset_137();
RemoteControlStart_137();

RemoteControlTempAdjust_137();












StartStopCommand_138();
StartStopStatus_138();
Alarm_138();
MalfunctionCode_138();




RoomTemp_138();
TempAdjust_138();
FilterSign_138();
FilterSignReset_138();
RemoteControlStart_138();

RemoteControlTempAdjust_138();












StartStopCommand_139();
StartStopStatus_139();
Alarm_139();
MalfunctionCode_139();




RoomTemp_139();
TempAdjust_139();
FilterSign_139();
FilterSignReset_139();
RemoteControlStart_139();

RemoteControlTempAdjust_139();












StartStopCommand_141();
StartStopStatus_141();
Alarm_141();
MalfunctionCode_141();




RoomTemp_141();
TempAdjust_141();
FilterSign_141();
FilterSignReset_141();
RemoteControlStart_141();

RemoteControlTempAdjust_141();












StartStopCommand_142();
StartStopStatus_142();
Alarm_142();
MalfunctionCode_142();




RoomTemp_142();
TempAdjust_142();
FilterSign_142();
FilterSignReset_142();
RemoteControlStart_142();

RemoteControlTempAdjust_142();












StartStopCommand_143();
StartStopStatus_143();
Alarm_143();
MalfunctionCode_143();




RoomTemp_143();
TempAdjust_143();
FilterSign_143();
FilterSignReset_143();
RemoteControlStart_143();

RemoteControlTempAdjust_143();












StartStopCommand_144();
StartStopStatus_144();
Alarm_144();
MalfunctionCode_144();




RoomTemp_144();
TempAdjust_144();
FilterSign_144();
FilterSignReset_144();
RemoteControlStart_144();

RemoteControlTempAdjust_144();












StartStopCommand_145();
StartStopStatus_145();
Alarm_145();
MalfunctionCode_145();




RoomTemp_145();
TempAdjust_145();
FilterSign_145();
FilterSignReset_145();
RemoteControlStart_145();

RemoteControlTempAdjust_145();












StartStopCommand_146();
StartStopStatus_146();
Alarm_146();
MalfunctionCode_146();




RoomTemp_146();
TempAdjust_146();
FilterSign_146();
FilterSignReset_146();
RemoteControlStart_146();

RemoteControlTempAdjust_146();












StartStopCommand_147();
StartStopStatus_147();
Alarm_147();
MalfunctionCode_147();




RoomTemp_147();
TempAdjust_147();
FilterSign_147();
FilterSignReset_147();
RemoteControlStart_147();

RemoteControlTempAdjust_147();












StartStopCommand_148();
StartStopStatus_148();
Alarm_148();
MalfunctionCode_148();




RoomTemp_148();
TempAdjust_148();
FilterSign_148();
FilterSignReset_148();
RemoteControlStart_148();

RemoteControlTempAdjust_148();












StartStopCommand_160();
StartStopStatus_160();
Alarm_160();
MalfunctionCode_160();




RoomTemp_160();
TempAdjust_160();
FilterSign_160();
FilterSignReset_160();
RemoteControlStart_160();

RemoteControlTempAdjust_160();












StartStopCommand_161();
StartStopStatus_161();
Alarm_161();
MalfunctionCode_161();




RoomTemp_161();
TempAdjust_161();
FilterSign_161();
FilterSignReset_161();
RemoteControlStart_161();

RemoteControlTempAdjust_161();












StartStopCommand_162();
StartStopStatus_162();
Alarm_162();
MalfunctionCode_162();




RoomTemp_162();
TempAdjust_162();
FilterSign_162();
FilterSignReset_162();
RemoteControlStart_162();

RemoteControlTempAdjust_162();












StartStopCommand_163();
StartStopStatus_163();
Alarm_163();
MalfunctionCode_163();




RoomTemp_163();
TempAdjust_163();
FilterSign_163();
FilterSignReset_163();
RemoteControlStart_163();

RemoteControlTempAdjust_163();












StartStopCommand_164();
StartStopStatus_164();
Alarm_164();
MalfunctionCode_164();




RoomTemp_164();
TempAdjust_164();
FilterSign_164();
FilterSignReset_164();
RemoteControlStart_164();

RemoteControlTempAdjust_164();












StartStopCommand_165();
StartStopStatus_165();
Alarm_165();
MalfunctionCode_165();




RoomTemp_165();
TempAdjust_165();
FilterSign_165();
FilterSignReset_165();
RemoteControlStart_165();

RemoteControlTempAdjust_165();












StartStopCommand_166();
StartStopStatus_166();
Alarm_166();
MalfunctionCode_166();




RoomTemp_166();
TempAdjust_166();
FilterSign_166();
FilterSignReset_166();
RemoteControlStart_166();

RemoteControlTempAdjust_166();












StartStopCommand_167();
StartStopStatus_167();
Alarm_167();
MalfunctionCode_167();




RoomTemp_167();
TempAdjust_167();
FilterSign_167();
FilterSignReset_167();
RemoteControlStart_167();

RemoteControlTempAdjust_167();












StartStopCommand_176();
StartStopStatus_176();
Alarm_176();
MalfunctionCode_176();




RoomTemp_176();
TempAdjust_176();
FilterSign_176();
FilterSignReset_176();
RemoteControlStart_176();

RemoteControlTempAdjust_176();












StartStopCommand_193();
StartStopStatus_193();
Alarm_193();
MalfunctionCode_193();




RoomTemp_193();
TempAdjust_193();
FilterSign_193();
FilterSignReset_193();
RemoteControlStart_193();

RemoteControlTempAdjust_193();












StartStopCommand_194();
StartStopStatus_194();
Alarm_194();
MalfunctionCode_194();




RoomTemp_194();
TempAdjust_194();
FilterSign_194();
FilterSignReset_194();
RemoteControlStart_194();

RemoteControlTempAdjust_194();












StartStopCommand_195();
StartStopStatus_195();
Alarm_195();
MalfunctionCode_195();




RoomTemp_195();
TempAdjust_195();
FilterSign_195();
FilterSignReset_195();
RemoteControlStart_195();

RemoteControlTempAdjust_195();












StartStopCommand_196();
StartStopStatus_196();
Alarm_196();
MalfunctionCode_196();




RoomTemp_196();
TempAdjust_196();
FilterSign_196();
FilterSignReset_196();
RemoteControlStart_196();

RemoteControlTempAdjust_196();












StartStopCommand_197();
StartStopStatus_197();
Alarm_197();
MalfunctionCode_197();




RoomTemp_197();
TempAdjust_197();
FilterSign_197();
FilterSignReset_197();
RemoteControlStart_197();

RemoteControlTempAdjust_197();












StartStopCommand_198();
StartStopStatus_198();
Alarm_198();
MalfunctionCode_198();




RoomTemp_198();
TempAdjust_198();
FilterSign_198();
FilterSignReset_198();
RemoteControlStart_198();

RemoteControlTempAdjust_198();












StartStopCommand_199();
StartStopStatus_199();
Alarm_199();
MalfunctionCode_199();




RoomTemp_199();
TempAdjust_199();
FilterSign_199();
FilterSignReset_199();
RemoteControlStart_199();

RemoteControlTempAdjust_199();












StartStopCommand_200();
StartStopStatus_200();
Alarm_200();
MalfunctionCode_200();




RoomTemp_200();
TempAdjust_200();
FilterSign_200();
FilterSignReset_200();
RemoteControlStart_200();

RemoteControlTempAdjust_200();












StartStopCommand_201();
StartStopStatus_201();
Alarm_201();
MalfunctionCode_201();




RoomTemp_201();
TempAdjust_201();
FilterSign_201();
FilterSignReset_201();
RemoteControlStart_201();

RemoteControlTempAdjust_201();












StartStopCommand_202();
StartStopStatus_202();
Alarm_202();
MalfunctionCode_202();




RoomTemp_202();
TempAdjust_202();
FilterSign_202();
FilterSignReset_202();
RemoteControlStart_202();

RemoteControlTempAdjust_202();












StartStopCommand_203();
StartStopStatus_203();
Alarm_203();
MalfunctionCode_203();




RoomTemp_203();
TempAdjust_203();
FilterSign_203();
FilterSignReset_203();
RemoteControlStart_203();

RemoteControlTempAdjust_203();












StartStopCommand_204();
StartStopStatus_204();
Alarm_204();
MalfunctionCode_204();




RoomTemp_204();
TempAdjust_204();
FilterSign_204();
FilterSignReset_204();
RemoteControlStart_204();

RemoteControlTempAdjust_204();












StartStopCommand_205();
StartStopStatus_205();
Alarm_205();
MalfunctionCode_205();




RoomTemp_205();
TempAdjust_205();
FilterSign_205();
FilterSignReset_205();
RemoteControlStart_205();

RemoteControlTempAdjust_205();












StartStopCommand_206();
StartStopStatus_206();
Alarm_206();
MalfunctionCode_206();




RoomTemp_206();
TempAdjust_206();
FilterSign_206();
FilterSignReset_206();
RemoteControlStart_206();

RemoteControlTempAdjust_206();












StartStopCommand_207();
StartStopStatus_207();
Alarm_207();
MalfunctionCode_207();




RoomTemp_207();
TempAdjust_207();
FilterSign_207();
FilterSignReset_207();
RemoteControlStart_207();

RemoteControlTempAdjust_207();












StartStopCommand_208();
StartStopStatus_208();
Alarm_208();
MalfunctionCode_208();




RoomTemp_208();
TempAdjust_208();
FilterSign_208();
FilterSignReset_208();
RemoteControlStart_208();

RemoteControlTempAdjust_208();












StartStopCommand_209();
StartStopStatus_209();
Alarm_209();
MalfunctionCode_209();




RoomTemp_209();
TempAdjust_209();
FilterSign_209();
FilterSignReset_209();
RemoteControlStart_209();

RemoteControlTempAdjust_209();












StartStopCommand_210();
StartStopStatus_210();
Alarm_210();
MalfunctionCode_210();




RoomTemp_210();
TempAdjust_210();
FilterSign_210();
FilterSignReset_210();
RemoteControlStart_210();

RemoteControlTempAdjust_210();












StartStopCommand_211();
StartStopStatus_211();
Alarm_211();
MalfunctionCode_211();




RoomTemp_211();
TempAdjust_211();
FilterSign_211();
FilterSignReset_211();
RemoteControlStart_211();

RemoteControlTempAdjust_211();












StartStopCommand_212();
StartStopStatus_212();
Alarm_212();
MalfunctionCode_212();




RoomTemp_212();
TempAdjust_212();
FilterSign_212();
FilterSignReset_212();
RemoteControlStart_212();

RemoteControlTempAdjust_212();












StartStopCommand_213();
StartStopStatus_213();
Alarm_213();
MalfunctionCode_213();




RoomTemp_213();
TempAdjust_213();
FilterSign_213();
FilterSignReset_213();
RemoteControlStart_213();

RemoteControlTempAdjust_213();












StartStopCommand_214();
StartStopStatus_214();
Alarm_214();
MalfunctionCode_214();




RoomTemp_214();
TempAdjust_214();
FilterSign_214();
FilterSignReset_214();
RemoteControlStart_214();

RemoteControlTempAdjust_214();












StartStopCommand_215();
StartStopStatus_215();
Alarm_215();
MalfunctionCode_215();




RoomTemp_215();
TempAdjust_215();
FilterSign_215();
FilterSignReset_215();
RemoteControlStart_215();

RemoteControlTempAdjust_215();












StartStopCommand_216();
StartStopStatus_216();
Alarm_216();
MalfunctionCode_216();




RoomTemp_216();
TempAdjust_216();
FilterSign_216();
FilterSignReset_216();
RemoteControlStart_216();

RemoteControlTempAdjust_216();












StartStopCommand_217();
StartStopStatus_217();
Alarm_217();
MalfunctionCode_217();




RoomTemp_217();
TempAdjust_217();
FilterSign_217();
FilterSignReset_217();
RemoteControlStart_217();

RemoteControlTempAdjust_217();












StartStopCommand_224();
StartStopStatus_224();
Alarm_224();
MalfunctionCode_224();




RoomTemp_224();
TempAdjust_224();
FilterSign_224();
FilterSignReset_224();
RemoteControlStart_224();

RemoteControlTempAdjust_224();












StartStopCommand_225();
StartStopStatus_225();
Alarm_225();
MalfunctionCode_225();




RoomTemp_225();
TempAdjust_225();
FilterSign_225();
FilterSignReset_225();
RemoteControlStart_225();

RemoteControlTempAdjust_225();












StartStopCommand_226();
StartStopStatus_226();
Alarm_226();
MalfunctionCode_226();




RoomTemp_226();
TempAdjust_226();
FilterSign_226();
FilterSignReset_226();
RemoteControlStart_226();

RemoteControlTempAdjust_226();












StartStopCommand_227();
StartStopStatus_227();
Alarm_227();
MalfunctionCode_227();




RoomTemp_227();
TempAdjust_227();
FilterSign_227();
FilterSignReset_227();
RemoteControlStart_227();

RemoteControlTempAdjust_227();












StartStopCommand_240();
StartStopStatus_240();
Alarm_240();
MalfunctionCode_240();




RoomTemp_240();
TempAdjust_240();
FilterSign_240();
FilterSignReset_240();
RemoteControlStart_240();

RemoteControlTempAdjust_240();












StartStopCommand_241();
StartStopStatus_241();
Alarm_241();
MalfunctionCode_241();




RoomTemp_241();
TempAdjust_241();
FilterSign_241();
FilterSignReset_241();
RemoteControlStart_241();

RemoteControlTempAdjust_241();












CL_Rejection_000();
SystemForcedOff_000();
CL_Rejection_064();
SystemForcedOff_064();
CL_Rejection_128();
SystemForcedOff_128();
CL_Rejection_192();
SystemForcedOff_192();

END_FUNCTION_BLOCK

(* stored: Version 1.1.0.1, ProductVersion 3.1.4024.12
   POU FB_BACnet_DAIKIN_MasterStation_III_No_1: Id {697b267d-405f-4f4d-8fce-d1cc2838ce8b}, SpecialFunc None *)
